PROGRAM MAIN
VAR
END_VAR

END_PROGRAM

(* stored: Version 1.1.0.1, ProductVersion 3.1.0.36
   POU MAIN: Id {f2e5b544-6944-45b4-9b5b-96de527ff477} *)
